{attribute 'qualified_only'}
{attribute 'strict'}
TYPE E_SA_SIM_CH_SM_STATE :
(
	IDLE := 0,
	CALIB,
	REF,
	MOV,
	STOP
);
END_TYPE

(* stored: Version 1.1.0.1, ProductVersion 3.1.4024.10
   DUT E_SA_SIM_CH_SM_STATE: Id {356272c5-0af8-4c40-b206-68e7404a8a94} *)
